// TIA Portal V20 export
VAR_GLOBAL   // PLC tag table "LGR_Const_SpeedSet"
END_VAR
VAR_GLOBAL CONSTANT   // user constants
   SPD_MANU_LL : USInt := 0;
   SPD_MANU_L : USInt := 1;   // SPD_JOG
   SPD_MANU_M : USInt := 2;   // POS_JOG
   SPD_AUTO_M : USInt := 3;
   SPD_AUTO_H : USInt := 4;
   SPD_HOME : USInt := 6;
   SPD_HOME_CREEP : USInt := 7;
   SPD_AUTO_CREEP : USInt := 5;
   SPD_FAULT : USInt := 8;
   SPD_FAULT_FAST : USInt := 9;
END_VAR
